(* IEC 61131-3 sources: astools/Data/ASTemplates/Default/Export Dialog/LogicalView/Libraries/AsArSdm, 2 files *)

(* ---- AsArSdm.var ---- *)
VAR CONSTANT
	sdmERR_NOT_EXIST			: UINT		:= 34900;	(*SDM not active*)
	sdmERR_ARREG				: UINT		:= 34901;	(*SDM AR registry error*)
	sdmERR_SYSTEMDUMP			: UINT		:= 34902;	(*SDM System dump error*)
	sdmERR_INVALID_DEVICE		: UINT		:= 34903;	(*SDM System dump invalid device*)
	sdmERR_INVALID_POINTER		: UINT		:= 34904;	(*SDM System dump invalid pointer*)
	sdmERR_INVALID_VALUE		: UINT		:= 34905;	(*SDM Invalid application mode*)
	sdmERR_OPTION_INVALID		: UINT		:= 34906;	(*SDM"Option" parameter invalid*)

	sdm_SYSTEMDUMP_PARAM		: UINT		:= 0;		(*SDM System Dump parameters only*)
	sdm_SYSTEMDUMP_DATA			: UINT		:= 1;		(*SDM SDM System Dump parameters and data files*)

	sdm_APPMODE_NOTUSED			: UINT		:= 0;		(*SDM Applicationmode not set*)
	sdm_APPMODE_OK				: UINT		:= 1;		(*SDM Application ok*)
	sdm_APPMODE_WARNING			: UINT		:= 2;		(*SDM Application warning *)
	sdm_APPMODE_ERROR			: UINT		:= 3;		(*SDM Application error*)

	sdmOPTION_NON_VOLATILE		: UDINT		:= 1;		(*permanently sets parameters*)
	sdmOPTION_VOLATILE			: UDINT		:= 0;		(*temporarily sets parameters*)
END_VAR

(* ---- AsArSdm.fun ---- *)
{REDUND_CONTEXT} {REDUND_UNREPLICABLE} FUNCTION_BLOCK SdmSystemDump			(*SDM - create a system dump; asynchronous execution*)
	VAR_INPUT
		enable			: BOOL;			(*enables execution*)
		configuration	: UDINT;		(*cfgSDM_SYSTEMDUMP_PARAM(0) parameters only or cfgSDM_SYSTEMDUMP_DATA(1) parameters and data-files*)
		pDevice			: UDINT;		(*Devicename given as a pointer*)
		pFile			: UDINT;		(*Filename given as a pointer*)
		pParam			: UDINT;		(*Parameterstring given as a pointer*)
	END_VAR

	VAR_OUTPUT
		status			: UINT;			(*execution status: ERR_OK, ERR_FUB_ENABLE_FALSE, ERR_FUB_BUSY, 0xXXXX = see help*)
	END_VAR

	VAR
        i_state			: UINT;			(*internal variable*)
		i_result		: UINT;			(*internal variable*)
        i_tmp			: UDINT;		(*internal variable*)
	END_VAR
END_FUNCTION_BLOCK

{REDUND_CONTEXT} {REDUND_UNREPLICABLE} FUNCTION_BLOCK SdmSetAppParam 	(*SDM - set application mode; asynchronous execution*)
	VAR_INPUT
		enable			: BOOL;			(*enables execution*)
		appMode			: UDINT;		(*cfgSDM_APPMODE_OK(1),cfgSDM_APPMODE_WARNING(2),cfgSDM_APPMODE_ERROR(3)*)
		pLink			: UDINT;		(*URL given as a pointer*)
		Option			: UDINT;		(*options: cfgOPTION_VOLATILE, cfgOPTION_NON_VOLATILE*)
	END_VAR

	VAR_OUTPUT
		status			: UINT;			(*execution status: ERR_OK, ERR_FUB_ENABLE_FALSE, ERR_FUB_BUSY, 0xXXXX = see help*)
	END_VAR

	VAR
        i_state			: UINT;			(*internal variable*)
		i_result		: UINT;			(*internal variable*)
        i_tmp			: UDINT;		(*internal variable*)
	END_VAR
END_FUNCTION_BLOCK
